Yaskawa INFORM job: R1_72,2(0,0)R2_MOD.JBI

/JOB
//NAME R1_72,2(0,0)R2_MOD
///FOLDERNAME KRIS-SCIANA
//POS
///NPOS 77,77,0,4,0,0
///TOOL 0
///POSTYPE PULSE
///PULSE
C00000=120729,38464,-23607,67702,92694,37114
C00001=130813,19897,-28859,40674,87554,31415
C00002=146503,13359,-34988,8933,69897,-84629
C00003=149406,-15453,-14205,34586,14154,-90922
C00004=162228,-76716,-47739,-17733,8035,-57819
C00005=116676,-56277,-93767,36796,58543,-83683
C00006=119975,-30594,-87710,23665,77906,-57976
C00007=119975,-31906,-87262,23741,77032,-58152
C00008=119975,-31304,-87473,23705,77435,-58070
C00009=121098,-31311,-87478,23052,77185,-57789
C00010=119855,-35918,-93693,23666,78800,-57828
C00011=130813,19897,-28859,40674,87554,31415
C00012=125083,56704,30738,54224,74995,24956
C00013=126358,57000,31561,53980,74051,25086
C00014=124721,62288,44734,63185,73473,22335
C00015=124721,62512,45919,63338,73183,22075
C00016=124721,62288,44734,63185,73473,22335
C00017=125305,62416,44881,63099,73087,22421
C00018=124721,62288,44734,63185,73473,22335
C00019=120729,38464,-23607,67702,92694,37114
C00020=120728,81583,44137,67576,84483,28591
C00021=120728,81594,44149,67576,84482,28590
C00022=120728,81598,44155,67576,84481,28590
C00023=121153,79204,40556,67418,84605,29065
C00024=121461,79214,40567,67348,84405,29106
C00025=121153,79204,40556,67418,84605,29065
C00026=120728,81598,44155,67576,84481,28590
C00027=120728,81522,44639,67599,84344,28446
C00028=120728,81417,45180,67625,84187,28282
C00029=120728,81522,44639,67599,84344,28446
C00030=120728,81598,44155,67576,84481,28590
C00031=120728,82318,42212,50838,72434,30029
C00032=120728,82713,44903,51184,71498,29492
C00033=120728,84371,46951,51284,71235,29340
C00034=120728,82713,44903,51184,71498,29492
C00035=120728,82318,42212,50838,72434,30029
C00036=120728,83470,39162,50303,74040,30931
C00037=120731,108704,30437,520,103146,-53106
C00038=120730,95364,30685,507,96140,-53135
C00039=120729,92856,31465,505,94371,-53142
C00040=120518,90602,30857,566,93586,-53206
C00041=120076,91948,31897,698,93643,-53342
C00042=120729,92386,31163,506,94315,-53143
C00043=120574,97951,39893,551,91803,-53198
C00044=121066,130208,79990,461,95227,-53028
C00045=121134,131914,82339,451,94657,-53008
C00046=120821,132587,79324,499,96860,-53101
C00047=120730,97149,30254,16854,109142,-86058
C00048=94374,59905,-24624,-6692,95808,-73268
C00049=94859,43835,-17383,-4554,74801,-71238
C00050=94859,41415,-16000,-4599,72712,-71159
C00051=88285,47130,-10285,7482,76539,-70280
C00052=94590,38531,-17304,-4457,72022,-71215
C00053=94826,41033,-16151,-4582,72608,-71165
C00054=88838,46898,-10539,7187,76531,-70115
C00055=90372,45128,-12368,6366,76638,-69653
C00056=101622,56236,-2911,-16255,82749,-70743
C00057=102210,62619,3889,-16550,81978,-70460
C00058=102039,71942,670,-16368,88461,-71374
C00059=120729,38464,-23607,67702,92694,37114
C00060=126358,57000,31561,53980,74051,25086
C00061=127340,53488,29402,53838,73202,25111
C00062=126552,50092,30148,59345,71642,24118
C00063=126411,61917,43233,59752,70711,23276
C00064=125699,61499,41475,59654,71606,23502
C00065=130813,19897,-28859,40674,87554,31415
C00066=146503,13359,-34988,8933,69897,-84629
C00067=149406,-15453,-14205,34586,14154,-90922
C00068=162228,-76716,-47739,-17733,8035,-57819
C00069=116676,-56277,-93767,36796,58543,-83683
C00070=119943,-37304,-91972,23749,77155,-58138
C00071=120915,-36130,-90230,23223,76506,-57981
C00072=120902,-23940,-82051,23132,77647,-57758
C00073=119420,-34845,-92709,23922,78850,-57946
C00074=130813,19897,-28859,40674,87554,31415
C00075=127963,-13691,-44237,56024,78067,29543
C00076=48492,61943,-11432,-541,72797,-1948
BC00000=247969,581384,1069855
BC00001=247969,581384,399097
BC00002=247968,581386,399096
BC00003=247968,581386,399096
BC00004=230897,482901,399096
BC00005=168206,509517,62465
BC00006=168206,509517,62465
BC00007=168206,509517,62465
BC00008=168206,509517,62465
BC00009=168206,509517,62465
BC00010=168206,509517,62465
BC00011=247969,581384,399097
BC00012=247969,581384,399097
BC00013=247969,581384,399097
BC00014=247969,581384,399097
BC00015=247969,581384,399097
BC00016=247969,581384,399097
BC00017=247969,581384,399097
BC00018=247969,581384,399097
BC00019=247969,581384,1069855
BC00020=247969,581384,1069855
BC00021=242395,578319,1053929
BC00022=240166,577093,1047559
BC00023=240163,576451,1029407
BC00024=240163,576451,1029407
BC00025=240163,576451,1029407
BC00026=240166,577093,1047559
BC00027=234047,579018,1046735
BC00028=234047,579018,1046735
BC00029=234047,579018,1046735
BC00030=240166,577093,1047559
BC00031=204016,615205,1075175
BC00032=204014,614569,1075175
BC00033=204014,614569,1075175
BC00034=204014,614569,1075175
BC00035=204016,615205,1075175
BC00036=222293,612873,1075175
BC00037=148834,597684,1075175
BC00038=148876,597689,1075175
BC00039=146152,596166,1075175
BC00040=145063,595557,1075175
BC00041=145063,595557,1075175
BC00042=145063,595557,1075175
BC00043=145063,595557,1075175
BC00044=145063,595557,1075175
BC00045=145063,595557,1075175
BC00046=145063,595557,1075175
BC00047=163962,558925,1075175
BC00048=16042,566310,1075175
BC00049=16207,572657,1075175
BC00050=16871,569169,1075175
BC00051=17137,567774,1075175
BC00052=17137,567774,1075175
BC00053=17137,567774,1075175
BC00054=17137,567774,1075175
BC00055=17137,567774,1075175
BC00056=17137,567774,1075175
BC00057=17137,567774,1075175
BC00058=17137,567774,1075175
BC00059=247969,581384,1069855
BC00060=247969,581384,399097
BC00061=247969,581384,399097
BC00062=247969,581384,399097
BC00063=247969,581384,399097
BC00064=247969,581384,399097
BC00065=247969,581384,399097
BC00066=247968,581386,399096
BC00067=247968,581386,399096
BC00068=230897,482901,399096
BC00069=168206,509517,62465
BC00070=168206,509517,62465
BC00071=168206,509517,62465
BC00072=168206,509517,62465
BC00073=168206,509517,62465
BC00074=247969,581384,399097
BC00075=247969,581384,399097
BC00076=49225,622868,1075175
///POSTYPE BASE
///RECTAN
///RCONF 0,0,0,0,1,0,0,0,0,0,0,0,0,0,0,0,0,0,0,0,0,0,0,0
P00006=2.006,1.622,-0.565,0.0000,0.0000,0.0000
P00021=0.073,2.058,-0.109,0.0000,0.0000,0.0000
///RCONF 0,0,0,0,0,0,0,0,0,0,0,0,0,0,0,0,0,0,0,0,0,0,0,0
P00030=-0.014,-0.768,0.131,0.0000,0.0000,0.0000
P00031=-0.170,0.039,-0.647,0.0000,0.0000,0.0000
//INST
///DATE 2025/04/29 11:03
///ATTR SC,RW
///GROUP1 RB1,BS1
NOP
'R2_72.2(0,0)
'Path S1184
SFTOF
MOVJ C00000 BC00000 VJ=100.00
MOVJ C00001 BC00001 VJ=100.00
MOVL C00002 BC00002 V=416.7
MOVL C00003 BC00003 V=416.7
MOVL C00004 BC00004 V=416.7
MOVL C00005 BC00005 V=416.7
MOVL C00006 BC00006 V=100.0
REFP 3 C00007 BC00007
CALL JOB:SEARCH-R1
SET P031 P006
SFTON P031
MOVL C00008 BC00008 V=100.0
REFP 3 C00009 BC00009
CALL JOB:SEARCH-R1
SET P031 P006
SFTON P031
MOVL C00010 BC00010 V=100.0
SFTOF
MOVJ C00011 BC00011 VJ=100.00
MOVJ C00012 BC00012 VJ=100.00
MOVL C00013 BC00013 V=166.7
MOVL C00014 BC00014 V=100.0
REFP 3 C00015 BC00015
CALL JOB:SEARCH-R1
SET P030 P006
SFTON P030
MOVL C00016 BC00016 V=100.0
REFP 3 C00017 BC00017
CALL JOB:SEARCH-R1
SET P030 P006
SFTON P030
MOVL C00018 BC00018 V=100.0
SFTOF
MOVJ C00019 BC00019 VJ=100.00
MOVJ C00020 BC00020 VJ=100.00
MOVL C00021 BC00021 V=100.0
MOVL C00022 BC00022 V=100.0
MOVL C00023 BC00023 V=60.0
REFP 3 C00024 BC00024
CALL JOB:SEARCH-R1
SET P021 P006
SFTON P021
MOVL C00025 BC00025 V=60.0
MOVL C00026 BC00026 V=100.0
MOVL C00027 BC00027 V=60.0
REFP 3 C00028 BC00028
CALL JOB:SEARCH-R1
SET P021 P006
SFTON P021
MOVL C00029 BC00029 V=60.0
MOVL C00030 BC00030 V=100.0
MOVL C00031 BC00031 V=100.0
MOVL C00032 BC00032 V=60.0
REFP 3 C00033 BC00033
CALL JOB:SEARCH-R1
SET P021 P006
SFTON P021
MOVL C00034 BC00034 V=60.0
MOVL C00035 BC00035 V=100.0
MOVL C00036 BC00036 V=100.0
'Path W1186
SFTOF
SFTON P021
MOVJ C00037 BC00037 VJ=100.00
MOVJ C00038 BC00038 VJ=100.00
MOVL C00039 BC00039 V=100.0
CALL JOB:COFNIJ_DRUT
MOVL C00040 BC00040 V=100.0 PL=0
REFP 1 C00041 BC00041
REFP 2 C00042 BC00042
MACRO1 MJ#(0) ARGF6
ARCON
MOVL C00043 BC00043 V=10.8
MOVL C00044 BC00044 V=10.8
MOVL C00045 BC00045 V=10.0
ARCOF
MOVL C00046 BC00046 V=100.0
MOVL C00047 BC00047 V=100.0
SFTOF
'Path W1188
SFTOF
SFTON P021
MOVJ C00048 BC00048 VJ=100.00
MOVJ C00049 BC00049 VJ=100.00
MOVJ C00050 BC00050 VJ=100.00
MOVL C00051 BC00051 V=100.0 PL=0
REFP 1 C00052 BC00052
REFP 2 C00053 BC00053
MACRO1 MJ#(0) ARGF6
ARCON
MOVL C00054 BC00054 V=8.3
MOVL C00055 BC00055 V=8.3
MOVL C00056 BC00056 V=8.3
MOVL C00057 BC00057 V=8.3
ARCOF
MOVL C00058 BC00058 V=100.0
SFTOF
MOVJ C00059 BC00059 VJ=100.00
MOVL C00060 BC00060 V=400.0
SFTON P030
MOVL C00061 BC00061 V=166.7
MOVL C00062 BC00062 V=100.0 PL=0
MACRO1 MJ#(0) ARGF7
ARCON
MOVL C00063 BC00063 V=9.2
ARCOF
MOVL C00064 BC00064 V=166.7
SFTOF
MOVJ C00065 BC00065 VJ=100.00
MOVL C00066 BC00066 V=416.7
MOVL C00067 BC00067 V=416.7
MOVL C00068 BC00068 V=416.7
MOVL C00069 BC00069 V=416.7
MOVL C00070 BC00070 V=100.0
SFTON P031
MACRO1 MJ#(0) ARGF6
MOVL C00071 BC00071 V=100.0 PL=0
ARCON
MOVL C00072 BC00072 V=11.7
ARCOF
MOVL C00073 BC00073 V=166.7
SFTOF
MOVJ C00074 BC00074 VJ=100.00
MOVJ C00075 BC00075 VJ=100.00
MOVJ C00076 BC00076 VJ=100.00
SFTOF
END
